{attribute 'GeneratedUsingTerminal: EK1100-0000-0018'}
{attribute addProperty BoxType "EK1100-0000-0018"}
{attribute addProperty Id "Beckhoff_EL29xxEK1122Beckhoff_EL29xxEK1122_F1BDF7ED2A_0001_EL2911_0000_0016EL2911_3424714D38A_0002_EL2912_0000_0016EL2912_BFF8CF1936"}
{attribute addProperty CRC "4240866116"}
{attribute addProperty Size "76"}
TYPE Beckhoff_EL29xx_FCC67B44 EXTENDS EK1100_1FC0878B :
STRUCT
	{attribute addProperty Name "Beckhoff_EL29xxEK1122"}
	Beckhoff_EL29xxEK1122 : Beckhoff_EL29xxEK1122_F1BDF7ED;
	{attribute addProperty Name "A_0001_EL2911_0000_0016"}
	A_0001_EL2911_0000_0016 : EL2911_3424714D;
	{attribute addProperty Name "A_0002_EL2912_0000_0016"}
	A_0002_EL2912_0000_0016 : EL2912_BFF8CF19;
END_STRUCT
END_TYPE

(* stored: Version 1.2.0.0, ProductVersion 3.1.4024.9
   DUT Beckhoff_EL29xx_FCC67B44: Id {2756ec35-7ef2-4e99-8bc9-2e052aa70c99} *)
